PROGRAM Read_Payload
VAR
	Payload_EMA	: REAL;
	Payload_Raw	: REAL;
	Payload		: REAL;
	
	Threshold	: REAL := 70;	
	Overload	: BOOL := FALSE;
END_VAR

(* raw & ema payload *)
Payload_EMA := Background_Payload.Payload_EMA;
Payload_Raw := Background_Payload.Payload;

(* get payload when stationary *)
//IF Inclination < 5 AND Tilt < 5 AND Speed < 1 THEN
	Payload	:= Background_Payload.Payload;
//END_IF

(* check for overload *)
IF Payload > Threshold THEN
	Overload := TRUE;
ELSE
	Overload := FALSE;	
END_IF

END_PROGRAM

(* stored: Version 1.1.0.1, ProductVersion 3.1.4024.6
   POU Read_Payload: Id {54a58c0d-9bb6-4287-ad4a-87a5313c1987}, SpecialFunc None *)
